(* CODESYS project IFTTT_V1.1.library
   Version: 1.1
   Author: Kurt Braun
   Title: IFTTT_Lib
   Placeholder: PlaceholderTemplate
   LanguageModelAttribute: qualified-access-only
   Company: Kurt Braun

Project tree, tasks and I/O mapping:
  libraries: SysTypes2 Interfaces, * (System); SysProcess, * (System); Standard, * (System)
  30 Visualizations/
  10 Documentation/
  80 Status/
  20 Program Organization Units/
    function curl_string [ST]
    function block IFTTT_Send [ST]
  00000000-0000-0000-0000-000000000000|D:\CoDeSys\LibrariesV3\trunk\Intern\CAA\CAA Template\3.4.0.0 draft\Placeholder.xml
  00000000-0000-0000-0000-000000000000|D:\CoDeSys\LibrariesV3\trunk\Intern\CAA\CAA Template\3.2.0.3 draft\Prefix.pdf
  00000000-0000-0000-0000-000000000000|D:\CoDeSys\LibrariesV3\trunk\Intern\CAA\CAA Template\3.5.2.0 draft\Placeholder.xml
*)

// 20 Program Organization Units/curl_string
FUNCTION curl_string : STRING(255)
VAR_INPUT
	sValue1 : STRING;
	sValue2 : STRING;
	sValue3 : STRING;
	sEvent : STRING := 'event';
	sKey : STRING := '123456789012345678901234';
END_VAR
VAR
	sHoldString: STRING(255);
END_VAR
(*
curl -X POST -H "Content-Type: application/json" -d "{\"value1\":\"Hello \",\"value2\":\"World \",\"value3\":\"!\"}" https://maker.ifttt.com/trigger/{email}/with/key/dScfmjG8sTQuYYjcgHrCCw -k
OR
curl -X POST https://maker.ifttt.com/trigger/{event}/with/key/dScfmjG8sTQuYYjcgHrCCw
*)

sHoldString := 'curl -X POST ';	
sHoldString := CONCAT(sHoldString, '-H "Content-Type: application/json" -d "{\"value1\":\"');
sHoldString := CONCAT(sHoldString, sValue1);
sHoldString := CONCAT(sHoldString, '\",\"value2\":\"');
sHoldString := CONCAT(sHoldString, sValue2);
sHoldString := CONCAT(sHoldString, '\",\"value3\":\"');
sHoldString := CONCAT(sHoldString, sValue3);	
sHoldString := CONCAT(sHoldString, '\"}" https://maker.ifttt.com/trigger/{');	
sHoldString := CONCAT(sHoldString, sEvent);	
sHoldString := CONCAT(sHoldString, '}/with/key/');	
sHoldString := CONCAT(sHoldString, sKey);	
sHoldString := CONCAT(sHoldString, ' -k');	
curl_string := sHoldString;

END_FUNCTION

// 20 Program Organization Units/IFTTT_Send
FUNCTION_BLOCK IFTTT_Send
VAR_INPUT 
	sValue1 : STRING;
	sValue2 : STRING;
	sValue3 : STRING;
	sEvent : STRING := 'event';
	sKey : STRING := '123456789012345678901234';
	xSend: BOOL;
END_VAR
VAR_OUTPUT
	xError : BOOL;
	xSent : BOOL;
	sReturn_String : STRING(255);
END_VAR
VAR
	sCommand_String : STRING(255);
	pResult : RTS_IEC_RESULT;
	GO_TRIG : R_TRIG;
	xSend_Once : BOOL;
END_VAR
// curl -X POST -H "Content-Type: application/json" -d "{\"value1\":\"Hello \",\"value2\":\"World \",\"value3\":\"!\"}" https://maker.ifttt.com/trigger/{email}/with/key/123456789012345678901234 -k

sCommand_String := curl_string(
	sValue1 := sValue1,
	sValue2 := sValue2,
	sValue3 := sValue3,
	sEvent := sEvent,
	sKey := sKey,
	);

GO_TRIG(CLK := xSend);
IF GO_TRIG.Q THEN
	xSend_Once := TRUE;
END_IF
		
IF xSend_Once THEN	
	SysProcessExecuteCommand2(pszCommand:=sCommand_String, pszStdOut := sReturn_String, udiStdOutLen := 255, pResult:= pResult);
	xSend_Once := FALSE;
END_IF

xError := FALSE;
xSent := FALSE;
//Error
IF (sReturn_String = 'Bad Request$N') OR (sReturn_String =  '{"errors":[{"message":"You sent an invalid key."}]}') THEN
	xError := TRUE;
	xSent := FALSE;
END_IF

//'Congratulations! You$'ve fired the email event'
IF (sReturn_String = 'Congratulations! You$'ve fired the email event') THEN
	xError := FALSE;
	xSent := TRUE;
END_IF

END_FUNCTION_BLOCK
